KUKA KRL program: welding_process.src, welding_process.dat

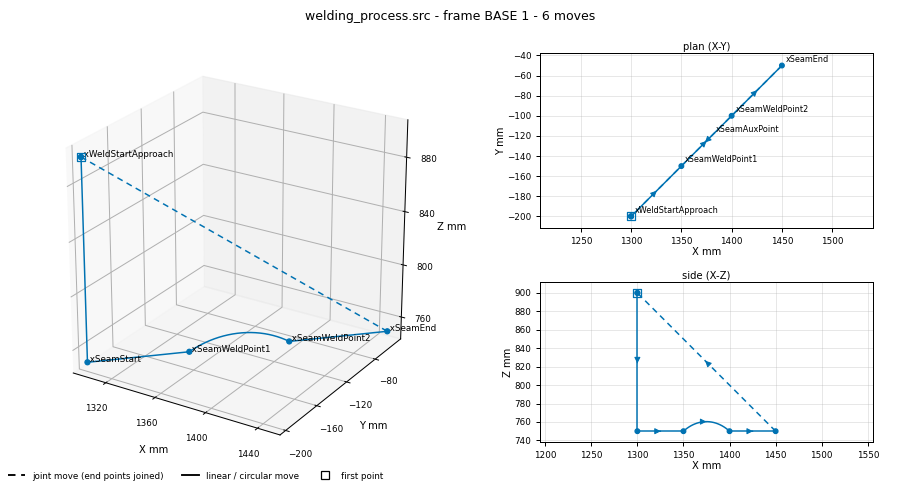
[picture p0: tool path of welding_process.src in frame BASE 1, 6 of 6 moves have a stored position in this frame; points joined in program order, loops and branches not executed]
--- welding_process.src ---
&ACCESS RVP
&REL 1
&COMMENT Modern Spline Arc Welding Routine
GLOBAL DEF welding_process()
  ; ========================================================
  ; ARC WELDING MOTION TRAJECTORY
  ; Tests: KSS 8.6+ Modern SPLINE blocks (SPLINE, SPTP, SLIN, SCIRC),
  ; Analog outputs ($ANOUT), Triggers and CodeLens references
  ; ========================================================
  BAS(#INITMOV, 0)
  $TOOL = TOOL_DATA[1]
  $BASE = BASE_DATA[1]

  ; Move to seam pre-position with Spline PTP
  SPTP xWeldStartApproach WITH $VEL_AXIS[1]=80

  ; Modern KSS continuous contour SPLINE block
  SPLINE
    SPL xSeamStart WITH $VEL.CP = 1.0
    SLIN xSeamWeldPoint1 WITH $VEL.CP = 0.65
    SCIRC xSeamAuxPoint, xSeamWeldPoint2 WITH $VEL.CP = 0.65
    SLIN xSeamEnd WITH $VEL.CP = 0.85
  ENDSPLINE

  ; Retract motion
  SPTP xWeldStartApproach WITH $VEL_AXIS[1]=90
END

--- welding_process.dat ---
&ACCESS RVP
&REL 1
DEFDAT welding_process
  DECL E6POS xWeldStartApproach = {X 1300.0, Y -200.0, Z 900.0, A 0.0, B 45.0, C 0.0, S 2, T 35}
  DECL E6POS xSeamStart = {X 1300.0, Y -200.0, Z 750.0, A 0.0, B 45.0, C 0.0, S 2, T 35}
  DECL E6POS xSeamWeldPoint1 = {X 1350.0, Y -150.0, Z 750.0, A 0.0, B 45.0, C 0.0, S 2, T 35}
  DECL E6POS xSeamAuxPoint = {X 1380.0, Y -120.0, Z 760.0, A 0.0, B 45.0, C 0.0, S 2, T 35}
  DECL E6POS xSeamWeldPoint2 = {X 1400.0, Y -100.0, Z 750.0, A 0.0, B 45.0, C 0.0, S 2, T 35}
  DECL E6POS xSeamEnd = {X 1450.0, Y -50.0, Z 750.0, A 0.0, B 45.0, C 0.0, S 2, T 35}
ENDDAT
